// Takes two input parameters, Code and Message, and returns an FsFB_Error object.
FUNCTION FsF_Error : REFERENCE TO FsFB_Error
VAR_INPUT
	Code : FsT_ErrCode;
	Message : FsT_ErrMsg;
END_VAR
VAR_STAT
	fbError : FsFB_ErrorDefinition;
END_VAR

CASE Code OF
	FsGVL_ErrorCodes.NO_ERROR: 
		fbError.Code := FsGVL_ErrorCodes.NO_ERROR;
		fbError.Message := 'No Error.';
ELSE
	fbError.Code :=	Code;
	fbError.Message := Message;
	END_CASE
FsF_Error REF= fbError;

END_FUNCTION

(* stored: Version 1.1.0.1, ProductVersion 3.1.4024.4
   POU FsF_Error: Id {4f691800-b13c-48a2-aabc-a2a5d345197f}, SpecialFunc None *)
